// TIA Portal V17 export
// export: Created 2024-08-07T21:44:00.6796067Z, ExportSetting WithDefaults, DisplayName Totally Integrated Automation Portal, DisplayVersion V17 Update 7, DisplayName TIA Portal Openness, DisplayVersion V17 Update 7, DisplayName TIA Portal Version Control Interface, DisplayVersion V17, DisplayName SINAMICS Startdrive Advanced, DisplayVersion V17 SP2, DisplayName SINAMICS Startdrive G110M, G120, G120C, G120D, G120P, G115D, DisplayVersion V17 SP2, DisplayName SINAMICS Startdrive G130, G150, S120, S150, SINAMICS MV, S210, DisplayVersion V17 SP2, DisplayName STEP 7 Professional, DisplayVersion V17 Update 7, DisplayName STEP 7 Safety, DisplayVersion V17 Update 6, DisplayName WinCC Advanced / Unified PC, DisplayVersion V17 Update 7
DATA_BLOCK "DB_DateTimeAndShifts_Instance"   // DB5010
VERSION : 0.1
// stored: AutoNumber false, DBAccessibleFromOPCUA true, DBAccessibleFromWebserver true, InstanceOfName FB_DateTimeAndShifts, InstanceOfType FB
"FB_DateTimeAndShifts"
   // VAR_INPUT
   //    iSettingsSecurity : Bool := TRUE;
   // END_VAR
   // VAR
   //    Edges : Struct
   //       Shift1Started : Bool := TRUE;
   //       Shift2Started : Bool := FALSE;
   //       Shift3Started : Bool := FALSE;
   //    END_STRUCT;
   // END_VAR
   // VAR RETAIN
   //    Settings : Struct
   //       Actual { S7_SetPoint := 'True'} : "UDT_DateTimeAndShiftsSettings";
   //       Last { S7_SetPoint := 'True'} : "UDT_DateTimeAndShiftsSettings";
   //       Status : Struct
   //          SettingsCanBeChanged : Bool := TRUE;
   //       END_STRUCT;
   //       Commands : Struct
   //          DateAndTimeUse : Bool := FALSE;
   //          DateAndTimeSet : Bool := FALSE;
   //       END_STRUCT;
   //    END_STRUCT;
   // END_VAR
   // VAR
   //    ActualValues : Struct
   //       DateAndTime : DTL := DTL#2023-02-15-10:23:05.248224204;
   //       DayOfYear : UInt := 46;
   //    END_STRUCT;
   //    ShiftStatus { S7_SetPoint := 'True'} : "UDT_ShiftStatus";
   //    TimeTransformationRule { S7_SetPoint := 'True'} : TimeTransformationRule;
   //    Set_timezone_results { ExternalAccessible := 'False'; ExternalVisible := 'False'; ExternalWritable := 'False'} : Struct
   //       done { ExternalAccessible := 'False'; ExternalVisible := 'False'; ExternalWritable := 'False'} : Bool;
   //       busy { ExternalAccessible := 'False'; ExternalVisible := 'False'; ExternalWritable := 'False'} : Bool;
   //       error { ExternalAccessible := 'False'; ExternalVisible := 'False'; ExternalWritable := 'False'} : Bool;
   //       status { ExternalAccessible := 'False'; ExternalVisible := 'False'; ExternalWritable := 'False'} : Word;
   //    END_STRUCT;
   // END_VAR
BEGIN
   Settings.Actual.DateAndTime := DTL#2019-01-17-00:00:00;
   Settings.Actual.Shift1Enabled := TRUE;
   Settings.Actual.Shift1StartTime := TOD#06:00:00;
   Settings.Actual.Shift1EndTime := TOD#14:00:00;
   Settings.Actual.Shift2Enabled := TRUE;
   Settings.Actual.Shift2StartTime := TOD#14:00:00;
   Settings.Actual.Shift2EndTime := TOD#22:00:00;
   Settings.Actual.Shift3Enabled := TRUE;
   Settings.Actual.Shift3StartTime := TOD#22:00:00;
   Settings.Actual.Shift3EndTime := TOD#06:00:00;
   Settings.Last.DateAndTime := DTL#2019-01-17-00:00:00;
   Settings.Last.Shift1Enabled := TRUE;
   Settings.Last.Shift1StartTime := TOD#06:00:00;
   Settings.Last.Shift1EndTime := TOD#14:00:00;
   Settings.Last.Shift2Enabled := TRUE;
   Settings.Last.Shift2StartTime := TOD#14:00:00;
   Settings.Last.Shift2EndTime := TOD#22:00:00;
   Settings.Last.Shift3Enabled := TRUE;
   Settings.Last.Shift3StartTime := TOD#22:00:00;
   Settings.Last.Shift3EndTime := TOD#06:00:00;
   ShiftStatus.ShiftNumber := 1;
   ShiftStatus.ShiftActive := TRUE;
   ShiftStatus.Shift1Started := FALSE;
   ShiftStatus.Shift2Started := FALSE;
   ShiftStatus.Shift3Started := FALSE;
END_DATA_BLOCK
